// TIA Portal V19 export
TYPE "LAF_typeSinaDiagData"
TITLE = LAF_typeSinaDiagData
// Diagnostic information of a SINAMICS
// stored: Access Published
   STRUCT
      sinaType { ExternalWritable := 'False'} : UInt;   // 0=NO_TYPE, 114=G120, 124=S120, 125=S120_EPOS, 220=S200, 221=S200_EPOS, 222=S210, 223=S210_EPOS
      controlWord { ExternalWritable := 'False'} : Word;   // PROFIdrive control word 1
      statusWord { ExternalWritable := 'False'} : Word;   // PROFIdrive status word 1
      telegramNo { ExternalWritable := 'False'} : UInt;   // PROFIdrive telegram number
      eposStatusWord1 { ExternalWritable := 'False'} : Word;   // EPOS status word 1
      eposStatusWord2 { ExternalWritable := 'False'} : Word;   // EPOS status word 2
      operatingDisplay { ExternalWritable := 'False'} : UInt;   // Operating display
      override { ExternalWritable := 'False'} : Real;   // Override
      posSetValue { ExternalWritable := 'False'} : Real;   // Position setpoint value
      posActValue { ExternalWritable := 'False'} : Real;   // Position actual value
      velSetValue { ExternalWritable := 'False'} : Real;   // Velocity setpoint value
      velActValue { ExternalWritable := 'False'} : Real;   // Velocity actual value
      lengthUnit { ExternalWritable := 'False'} : Int;   // Length unit
      velocityUnit { ExternalWritable := 'False'} : Int;   // Velocity unit
      residualDistance { ExternalWritable := 'False'} : Real;   // Residual distance
      followingError { ExternalWritable := 'False'} : Real;   // Actual following error
      posControlWord { ExternalWritable := 'False'} : Word;   // PROFIdrive positioning control word 1
      posStatusWord { ExternalWritable := 'False'} : Word;   // PROFIdrive positioning status word 1
      blockSelected { ExternalWritable := 'False'} : Int;   // Selected transversing block
      blockActive { ExternalWritable := 'False'} : Int;   // Active transversing block
      mdiPosSetValue { ExternalWritable := 'False'} : Real;   // MDI position setpoint value
      faultCode { ExternalWritable := 'False'} : Array[0..7] of Word;   // Fault code 0..7
      alarmCode { ExternalWritable := 'False'} : Array[0..3] of Word;   // Alarm code 0..3
      speedSetValue { ExternalWritable := 'False'} : Real;   // Speed set value
      speedActValue { ExternalWritable := 'False'} : Real;   // Speed actual value
      safetyStatusWord { ExternalWritable := 'False'} : Word;   // Safety staus word
   END_STRUCT;
END_TYPE
